FUNCTION_BLOCK AMP4330 
VAR_INPUT
END_VAR
VAR_OUTPUT
END_VAR
VAR
END_VAR

END_FUNCTION_BLOCK

(* stored: Version 1.1.0.1, ProductVersion 3.1.4024.12
   POU AMP4330: Id {b332215d-2169-486d-a2bd-2d78fe8264ff}, SpecialFunc None *)
